PROGRAM MAIN
VAR
END_VAR

END_PROGRAM

(* stored: Version 1.1.0.1
   POU MAIN: Id {cabbfd91-7b70-4f1d-9791-779ee39410af} *)
